{attribute 'linkalways'} 
{attribute 'no_explicit_call' := 'This FB is a CLASS and must be accessed using methods or properties'}
{attribute 'enable_dynamic_creation'}
FUNCTION_BLOCK FINAL OR_DINT EXTENDS Node
VAR
	in1 : _DINT(0);
	in2 : _DINT(0);
	out : _DINT(0);
END_VAR

METHOD PUBLIC Clone : I_Node
VAR
	pNode : POINTER TO OR_DINT;
END_VAR
pNode := __NEW(OR_DINT);
Clone := pNode^;
END_METHOD

METHOD FB_init : BOOL
VAR_INPUT
	bInitRetains : BOOL; // if TRUE, the retain variables are initialized (warm start / cold start)
	bInCopyCode : BOOL;  // if TRUE, the instance afterwards gets moved into the copy code (online change)
END_VAR
AddInput('in1',THIS^.in1);
AddInput('in2',THIS^.in2);
AddOutput('out', THIS^.out);
END_METHOD

METHOD PROTECTED OnExecute
VAR
END_VAR
out.Value := in1.Value OR in2.Value;
END_METHOD

END_FUNCTION_BLOCK

(* stored: Version 1.1.0.1, ProductVersion 3.1.4024.15
   POU OR_DINT: Id {9dddc7ae-43b1-4da1-a420-498f00c9bdb1}, SpecialFunc None
   Folder Constructor: Id {81e984b5-9155-4f46-a8a1-7737f2c9bbc4}
   Method Clone: Id {c8c0918e-2ed5-4ba7-98fb-8749c03b0c4f}
   Method FB_init: Id {c80babb3-52fb-467b-b926-817db8cfe1c0}
   Method OnExecute: Id {22a3a7b6-f94a-48ac-97e4-0613fe3c33ee} *)
